TYPE ST_SaMElementModes :
STRUCT
	 fbUndefined							: FB_SaMElementNotAllowed;
     fbProduction							: FB_SaMElementProduction;
     fbMaintenance							: FB_SaMElementMaintenance;
     fbManual								: FB_SaMElementManual;
     fbWashing								: FB_SaMElementWashing;
	 fbDiagnostics							: FB_SaMElementDiagnostics;
END_STRUCT
END_TYPE

(* stored: Version 1.1.0.1
   DUT ST_SaMElementModes: Id {2d59ec36-1fc5-0744-26c1-8077eec3f922} *)
